	X =  365.642  mm,	Y =   -78.945  mm,	Z =   -251.457  mm,
	W =  90.000 deg,	P =   0.000 deg,	R =   90.000 deg
};
P[3235]{
   GP1:
	UF : 0, UT : 6,		CONFIG : 'N U T, 0, 0, 0',
	X =  364.632  mm,	Y =   -78.307  mm,	Z =   -251.452  mm,
	W =  90.000 deg,	P =   0.000 deg,	R =   90.000 deg
};
P[3236]{
   GP1:
	UF : 0, UT : 6,		CONFIG : 'N U T, 0, 0, 0',
	X =  359.937  mm,	Y =   -76.604  mm,	Z =   -251.287  mm,
	W =  90.000 deg,	P =   0.000 deg,	R =   90.000 deg
};
P[3237]{
   GP1:
	UF : 0, UT : 6,		CONFIG : 'N U T, 0, 0, 0',
	X =  357.838  mm,	Y =   -76.355  mm,	Z =   -251.028  mm,
	W =  90.000 deg,	P =   0.000 deg,	R =   90.000 deg
};
P[3238]{
   GP1:
	UF : 0, UT : 6,		CONFIG : 'N U T, 0, 0, 0',
	X =  355.930  mm,	Y =   -76.626  mm,	Z =   -251.285  mm,
	W =  90.000 deg,	P =   0.000 deg,	R =   90.000 deg
};
P[3239]{
   GP1:
	UF : 0, UT : 6,		CONFIG : 'N U T, 0, 0, 0',
	X =  353.780  mm,	Y =   -77.047  mm,	Z =   -251.080  mm,
	W =  90.000 deg,	P =   0.000 deg,	R =   90.000 deg
};
P[3240]{
   GP1:
	UF : 0, UT : 6,		CONFIG : 'N U T, 0, 0, 0',
	X =  353.192  mm,	Y =   -77.362  mm,	Z =   -251.275  mm,
	W =  90.000 deg,	P =   0.000 deg,	R =   90.000 deg
};
P[3241]{
   GP1:
	UF : 0, UT : 6,		CONFIG : 'N U T, 0, 0, 0',
	X =  352.107  mm,	Y =   -77.912  mm,	Z =   -251.405  mm,
	W =  90.000 deg,	P =   0.000 deg,	R =   90.000 deg
};
P[3242]{
   GP1:
	UF : 0, UT : 6,		CONFIG : 'N U T, 0, 0, 0',
	X =  349.503  mm,	Y =   -79.254  mm,	Z =   -251.336  mm,
	W =  90.000 deg,	P =   0.000 deg,	R =   90.000 deg
};
P[3243]{
   GP1:
	UF : 0, UT : 6,		CONFIG : 'N U T, 0, 0, 0',
	X =  346.830  mm,	Y =   -80.833  mm,	Z =   -251.422  mm,
	W =  90.000 deg,	P =   0.000 deg,	R =   90.000 deg
};
P[3244]{
   GP1:
	UF : 0, UT : 6,		CONFIG : 'N U T, 0, 0, 0',
	X =  345.177  mm,	Y =   -81.811  mm,	Z =   -251.480  mm,
	W =  90.000 deg,	P =   0.000 deg,	R =   90.000 deg
};
P[3245]{
   GP1:
	UF : 0, UT : 6,		CONFIG : 'N U T, 0, 0, 0',
	X =  342.562  mm,	Y =   -83.180  mm,	Z =   -251.136  mm,
	W =  90.000 deg,	P =   0.000 deg,	R =   90.000 deg
};
P[3246]{
   GP1:
	UF : 0, UT : 6,		CONFIG : 'N U T, 0, 0, 0',
	X =  337.354  mm,	Y =   -86.298  mm,	Z =   -251.409  mm,
	W =  90.000 deg,	P =   0.000 deg,	R =   90.000 deg
};
P[3247]{
   GP1:
	UF : 0, UT : 6,		CONFIG : 'N U T, 0, 0, 0',
	X =  336.571  mm,	Y =   -86.625  mm,	Z =   -251.103  mm,
	W =  90.000 deg,	P =   0.000 deg,	R =   90.000 deg
};
P[3248]{
   GP1:
	UF : 0, UT : 6,		CONFIG : 'N U T, 0, 0, 0',
	X =  335.626  mm,	Y =   -87.310  mm,	Z =   -251.441  mm,
	W =  90.000 deg,	P =   0.000 deg,	R =   90.000 deg
};
P[3249]{
   GP1:
	UF : 0, UT : 6,		CONFIG : 'N U T, 0, 0, 0',
	X =  334.747  mm,	Y =   -87.679  mm,	Z =   -251.108  mm,
	W =  90.000 deg,	P =   0.000 deg,	R =   90.000 deg
};
P[3250]{
   GP1:
	UF : 0, UT : 6,		CONFIG : 'N U T, 0, 0, 0',
	X =  332.760  mm,	Y =   -88.868  mm,	Z =   -251.208  mm,
	W =  90.000 deg,	P =   0.000 deg,	R =   90.000 deg
};
P[3251]{
   GP1:
	UF : 0, UT : 6,		CONFIG : 'N U T, 0, 0, 0',
	X =  332.024  mm,	Y =   -89.291  mm,	Z =   -251.201  mm,
	W =  90.000 deg,	P =   0.000 deg,	R =   90.000 deg
};
P[3252]{
   GP1:
	UF : 0, UT : 6,		CONFIG : 'N U T, 0, 0, 0',
	X =  326.457  mm,	Y =   -92.567  mm,	Z =   -251.352  mm,
	W =  90.000 deg,	P =   0.000 deg,	R =   90.000 deg
};
P[3253]{
   GP1:
	UF : 0, UT : 6,		CONFIG : 'N U T, 0, 0, 0',
	X =  323.513  mm,	Y =   -94.171  mm,	Z =   -251.117  mm,
	W =  90.000 deg,	P =   0.000 deg,	R =   90.000 deg
};
P[3254]{
   GP1:
	UF : 0, UT : 6,		CONFIG : 'N U T, 0, 0, 0',
	X =  318.378  mm,	Y =   -97.275  mm,	Z =   -251.456  mm,
	W =  90.000 deg,	P =   0.000 deg,	R =   90.000 deg
};
P[3255]{
   GP1:
	UF : 0, UT : 6,		CONFIG : 'N U T, 0, 0, 0',
	X =  317.185  mm,	Y =   -97.859  mm,	Z =   -251.203  mm,
	W =  90.000 deg,	P =   0.000 deg,	R =   90.000 deg
};
P[3256]{
   GP1:
	UF : 0, UT : 6,		CONFIG : 'N U T, 0, 0, 0',
	X =  316.114  mm,	Y =   -98.543  mm,	Z =   -251.361  mm,
	W =  90.000 deg,	P =   0.000 deg,	R =   90.000 deg
};
P[3257]{
   GP1:
	UF : 0, UT : 6,		CONFIG : 'N U T, 0, 0, 0',
	X =  314.155  mm,	Y =   -99.553  mm,	Z =   -251.068  mm,
	W =  90.000 deg,	P =   0.000 deg,	R =   90.000 deg
};
P[3258]{
   GP1:
	UF : 0, UT : 6,		CONFIG : 'N U T, 0, 0, 0',
	X =  313.148  mm,	Y =   -100.225  mm,	Z =   -251.288  mm,
	W =  90.000 deg,	P =   0.000 deg,	R =   90.000 deg
};
P[3259]{
   GP1:
	UF : 0, UT : 6,		CONFIG : 'N U T, 0, 0, 0',
	X =  310.503  mm,	Y =   -101.793  mm,	Z =   -251.386  mm,
	W =  90.000 deg,	P =   0.000 deg,	R =   90.000 deg
};
P[3260]{
   GP1:
	UF : 0, UT : 6,		CONFIG : 'N U T, 0, 0, 0',
	X =  309.548  mm,	Y =   -102.306  mm,	Z =   -251.294  mm,
	W =  90.000 deg,	P =   0.000 deg,	R =   90.000 deg
};
P[3261]{
   GP1:
	UF : 0, UT : 6,		CONFIG : 'N U T, 0, 0, 0',
	X =  306.446  mm,	Y =   -104.089  mm,	Z =   -251.273  mm,
	W =  90.000 deg,	P =   0.000 deg,	R =   90.000 deg
};
P[3262]{
   GP1:
	UF : 0, UT : 6,		CONFIG : 'N U T, 0, 0, 0',
	X =  303.476  mm,	Y =   -105.784  mm,	Z =   -251.224  mm,
	W =  90.000 deg,	P =   0.000 deg,	R =   90.000 deg
};
P[3263]{
   GP1:
	UF : 0, UT : 6,		CONFIG : 'N U T, 0, 0, 0',
	X =  302.259  mm,	Y =   -106.421  mm,	Z =   -251.065  mm,
	W =  90.000 deg,	P =   0.000 deg,	R =   90.000 deg
};
P[3264]{
   GP1:
	UF : 0, UT : 6,		CONFIG : 'N U T, 0, 0, 0',
	X =  301.391  mm,	Y =   -107.018  mm,	Z =   -251.300  mm,
	W =  90.000 deg,	P =   0.000 deg,	R =   90.000 deg
};
P[3265]{
   GP1:
	UF : 0, UT : 6,		CONFIG : 'N U T, 0, 0, 0',
	X =  298.634  mm,	Y =   -108.624  mm,	Z =   -251.331  mm,
	W =  90.000 deg,	P =   0.000 deg,	R =   90.000 deg
};
P[3266]{
   GP1:
	UF : 0, UT : 6,		CONFIG : 'N U T, 0, 0, 0',
	X =  297.240  mm,	Y =   -109.333  mm,	Z =   -251.101  mm,
	W =  90.000 deg,	P =   0.000 deg,	R =   90.000 deg
};
P[3267]{
   GP1:
	UF : 0, UT : 6,		CONFIG : 'N U T, 0, 0, 0',
	X =  295.855  mm,	Y =   -110.282  mm,	Z =   -251.463  mm,
	W =  90.000 deg,	P =   0.000 deg,	R =   90.000 deg
};
P[3268]{
   GP1:
	UF : 0, UT : 6,		CONFIG : 'N U T, 0, 0, 0',
	X =  295.155  mm,	Y =   -110.620  mm,	Z =   -251.300  mm,
	W =  90.000 deg,	P =   0.000 deg,	R =   90.000 deg
};
P[3269]{
   GP1:
	UF : 0, UT : 6,		CONFIG : 'N U T, 0, 0, 0',
	X =  294.447  mm,	Y =   -111.014  mm,	Z =   -251.266  mm,
	W =  90.000 deg,	P =   0.000 deg,	R =   90.000 deg
};
P[3270]{
   GP1:
	UF : 0, UT : 6,		CONFIG : 'N U T, 0, 0, 0',
	X =  293.600  mm,	Y =   -111.593  mm,	Z =   -251.484  mm,
	W =  90.000 deg,	P =   0.000 deg,	R =   90.000 deg
};
P[3271]{
   GP1:
	UF : 0, UT : 6,		CONFIG : 'N U T, 0, 0, 0',
	X =  291.360  mm,	Y =   -112.706  mm,	Z =   -251.045  mm,
	W =  90.000 deg,	P =   0.000 deg,	R =   90.000 deg
};
P[3272]{
   GP1:
	UF : 0, UT : 6,		CONFIG : 'N U T, 0, 0, 0',
	X =  289.173  mm,	Y =   -114.076  mm,	Z =   -251.307  mm,
	W =  90.000 deg,	P =   0.000 deg,	R =   90.000 deg
};
P[3273]{
   GP1:
	UF : 0, UT : 6,		CONFIG : 'N U T, 0, 0, 0',
	X =  287.782  mm,	Y =   -114.866  mm,	Z =   -251.275  mm,
	W =  90.000 deg,	P =   0.000 deg,	R =   90.000 deg
};
P[3274]{
   GP1:
	UF : 0, UT : 6,		CONFIG : 'N U T, 0, 0, 0',
	X =  285.771  mm,	Y =   -116.071  mm,	Z =   -251.381  mm,
	W =  90.000 deg,	P =   0.000 deg,	R =   90.000 deg
};
P[3275]{
   GP1:
	UF : 0, UT : 6,		CONFIG : 'N U T, 0, 0, 0',
	X =  283.058  mm,	Y =   -117.627  mm,	Z =   -251.356  mm,
	W =  90.000 deg,	P =   0.000 deg,	R =   90.000 deg
};
P[3276]{
   GP1:
	UF : 0, UT : 6,		CONFIG : 'N U T, 0, 0, 0',
	X =  282.254  mm,	Y =   -118.089  mm,	Z =   -251.350  mm,
	W =  90.000 deg,	P =   0.000 deg,	R =   90.000 deg
};
P[3277]{
   GP1:
	UF : 0, UT : 6,		CONFIG : 'N U T, 0, 0, 0',
	X =  279.242  mm,	Y =   -119.866  mm,	Z =   -251.442  mm,
	W =  90.000 deg,	P =   0.000 deg,	R =   90.000 deg
};
P[3278]{
   GP1:
	UF : 0, UT : 6,		CONFIG : 'N U T, 0, 0, 0',
	X =  277.448  mm,	Y =   -120.879  mm,	Z =   -251.386  mm,
	W =  90.000 deg,	P =   0.000 deg,	R =   90.000 deg
};
P[3279]{
   GP1:
	UF : 0, UT : 6,		CONFIG : 'N U T, 0, 0, 0',
	X =  276.850  mm,	Y =   -121.103  mm,	Z =   -251.091  mm,
	W =  90.000 deg,	P =   0.000 deg,	R =   90.000 deg
};
P[3280]{
   GP1:
	UF : 0, UT : 6,		CONFIG : 'N U T, 0, 0, 0',
	X =  275.892  mm,	Y =   -121.675  mm,	Z =   -251.138  mm,
	W =  90.000 deg,	P =   0.000 deg,	R =   90.000 deg
};
P[3281]{
   GP1:
	UF : 0, UT : 6,		CONFIG : 'N U T, 0, 0, 0',
	X =  272.785  mm,	Y =   -123.489  mm,	Z =   -251.187  mm,
	W =  90.000 deg,	P =   0.000 deg,	R =   90.000 deg
};
P[3282]{
   GP1:
	UF : 0, UT : 6,		CONFIG : 'N U T, 0, 0, 0',
	X =  270.250  mm,	Y =   -124.968  mm,	Z =   -251.224  mm,
	W =  90.000 deg,	P =   0.000 deg,	R =   90.000 deg
};
P[3283]{
   GP1:
	UF : 0, UT : 6,		CONFIG : 'N U T, 0, 0, 0',
	X =  267.856  mm,	Y =   -126.325  mm,	Z =   -251.164  mm,
	W =  90.000 deg,	P =   0.000 deg,	R =   90.000 deg
};
P[3284]{
   GP1:
	UF : 0, UT : 6,		CONFIG : 'N U T, 0, 0, 0',
	X =  266.892  mm,	Y =   -126.881  mm,	Z =   -251.161  mm,
	W =  90.000 deg,	P =   0.000 deg,	R =   90.000 deg
};
P[3285]{
   GP1:
	UF : 0, UT : 6,		CONFIG : 'N U T, 0, 0, 0',
	X =  265.651  mm,	Y =   -127.610  mm,	Z =   -251.192  mm,
	W =  90.000 deg,	P =   0.000 deg,	R =   90.000 deg
};
P[3286]{
   GP1:
	UF : 0, UT : 6,		CONFIG : 'N U T, 0, 0, 0',
	X =  262.122  mm,	Y =   -129.745  mm,	Z =   -251.428  mm,
	W =  90.000 deg,	P =   0.000 deg,	R =   90.000 deg
};
P[3287]{
   GP1:
	UF : 0, UT : 6,		CONFIG : 'N U T, 0, 0, 0',
	X =  257.854  mm,	Y =   -132.149  mm,	Z =   -251.281  mm,
	W =  90.000 deg,	P =   0.000 deg,	R =   90.000 deg
};
P[3288]{
   GP1:
	UF : 0, UT : 6,		CONFIG : 'N U T, 0, 0, 0',
	X =  256.892  mm,	Y =   -132.728  mm,	Z =   -251.340  mm,
	W =  90.000 deg,	P =   0.000 deg,	R =   90.000 deg
};
P[3289]{
   GP1:
	UF : 0, UT : 6,		CONFIG : 'N U T, 0, 0, 0',
	X =  256.166  mm,	Y =   -133.205  mm,	Z =   -251.481  mm,
	W =  90.000 deg,	P =   0.000 deg,	R =   90.000 deg
};
P[3290]{
   GP1:
	UF : 0, UT : 6,		CONFIG : 'N U T, 0, 0, 0',
	X =  251.767  mm,	Y =   -135.749  mm,	Z =   -251.492  mm,
	W =  90.000 deg,	P =   0.000 deg,	R =   90.000 deg
};
P[3291]{
   GP1:
	UF : 0, UT : 6,		CONFIG : 'N U T, 0, 0, 0',
	X =  249.950  mm,	Y =   -136.758  mm,	Z =   -251.391  mm,
	W =  90.000 deg,	P =   0.000 deg,	R =   90.000 deg
};
P[3292]{
   GP1:
	UF : 0, UT : 6,		CONFIG : 'N U T, 0, 0, 0',
	X =  248.916  mm,	Y =   -137.229  mm,	Z =   -251.087  mm,
	W =  90.000 deg,	P =   0.000 deg,	R =   90.000 deg
};
P[3293]{
   GP1:
	UF : 0, UT : 6,		CONFIG : 'N U T, 0, 0, 0',
	X =  244.453  mm,	Y =   -139.858  mm,	Z =   -251.213  mm,
	W =  90.000 deg,	P =   0.000 deg,	R =   90.000 deg
};
P[3294]{
   GP1:
	UF : 0, UT : 6,		CONFIG : 'N U T, 0, 0, 0',
	X =  241.068  mm,	Y =   -141.906  mm,	Z =   -251.440  mm,
	W =  90.000 deg,	P =   0.000 deg,	R =   90.000 deg
};
P[3295]{
   GP1:
	UF : 0, UT : 6,		CONFIG : 'N U T, 0, 0, 0',
	X =  239.719  mm,	Y =   -142.513  mm,	Z =   -251.022  mm,
	W =  90.000 deg,	P =   0.000 deg,	R =   90.000 deg
};
P[3296]{
   GP1:
	UF : 0, UT : 6,		CONFIG : 'N U T, 0, 0, 0',
	X =  234.349  mm,	Y =   -145.704  mm,	Z =   -251.240  mm,
	W =  90.000 deg,	P =   0.000 deg,	R =   90.000 deg
};
P[3297]{
   GP1:
	UF : 0, UT : 6,		CONFIG : 'N U T, 0, 0, 0',
	X =  230.397  mm,	Y =   -148.015  mm,	Z =   -251.313  mm,
	W =  90.000 deg,	P =   0.000 deg,	R =   90.000 deg
};
P[3298]{
   GP1:
	UF : 0, UT : 6,		CONFIG : 'N U T, 0, 0, 0',
	X =  229.049  mm,	Y =   -148.679  mm,	Z =   -251.034  mm,
	W =  90.000 deg,	P =   0.000 deg,	R =   90.000 deg
};
P[3299]{
   GP1:
	UF : 0, UT : 6,		CONFIG : 'N U T, 0, 0, 0',
	X =  226.182  mm,	Y =   -150.383  mm,	Z =   -251.153  mm,
	W =  90.000 deg,	P =   0.000 deg,	R =   90.000 deg
};
P[3300]{
   GP1:
	UF : 0, UT : 6,		CONFIG : 'N U T, 0, 0, 0',
	X =  222.300  mm,	Y =   -152.731  mm,	Z =   -251.410  mm,
	W =  90.000 deg,	P =   0.000 deg,	R =   90.000 deg
};
P[3301]{
   GP1:
	UF : 0, UT : 6,		CONFIG : 'N U T, 0, 0, 0',
	X =  220.364  mm,	Y =   -153.720  mm,	Z =   -251.098  mm,
	W =  90.000 deg,	P =   0.000 deg,	R =   90.000 deg
};
P[3302]{
   GP1:
	UF : 0, UT : 6,		CONFIG : 'N U T, 0, 0, 0',
	X =  218.957  mm,	Y =   -154.647  mm,	Z =   -251.377  mm,
	W =  90.000 deg,	P =   0.000 deg,	R =   90.000 deg
};
P[3303]{
   GP1:
	UF : 0, UT : 6,		CONFIG : 'N U T, 0, 0, 0',
	X =  214.839  mm,	Y =   -156.990  mm,	Z =   -251.293  mm,
	W =  90.000 deg,	P =   0.000 deg,	R =   90.000 deg
};
P[3304]{
   GP1:
	UF : 0, UT : 6,		CONFIG : 'N U T, 0, 0, 0',
	X =  213.334  mm,	Y =   -157.757  mm,	Z =   -251.045  mm,
	W =  90.000 deg,	P =   0.000 deg,	R =   90.000 deg
};
P[3305]{
   GP1:
	UF : 0, UT : 6,		CONFIG : 'N U T, 0, 0, 0',
	X =  209.437  mm,	Y =   -160.137  mm,	Z =   -251.362  mm,
	W =  90.000 deg,	P =   0.000 deg,	R =   90.000 deg
};
P[3306]{
   GP1:
	UF : 0, UT : 6,		CONFIG : 'N U T, 0, 0, 0',
	X =  205.579  mm,	Y =   -162.285  mm,	Z =   -251.166  mm,
	W =  90.000 deg,	P =   0.000 deg,	R =   90.000 deg
};
P[3307]{
   GP1:
	UF : 0, UT : 6,		CONFIG : 'N U T, 0, 0, 0',
	X =  204.500  mm,	Y =   -163.043  mm,	Z =   -251.494  mm,
	W =  90.000 deg,	P =   0.000 deg,	R =   90.000 deg
};
P[3308]{
   GP1:
	UF : 0, UT : 6,		CONFIG : 'N U T, 0, 0, 0',
	X =  203.455  mm,	Y =   -163.573  mm,	Z =   -251.316  mm,
	W =  90.000 deg,	P =   0.000 deg,	R =   90.000 deg
};
P[3309]{
   GP1:
	UF : 0, UT : 6,		CONFIG : 'N U T, 0, 0, 0',
	X =  202.079  mm,	Y =   -164.250  mm,	Z =   -251.032  mm,
	W =  90.000 deg,	P =   0.000 deg,	R =   90.000 deg
};
P[3310]{
   GP1:
	UF : 0, UT : 6,		CONFIG : 'N U T, 0, 0, 0',
	X =  199.549  mm,	Y =   -165.840  mm,	Z =   -251.344  mm,
	W =  90.000 deg,	P =   0.000 deg,	R =   90.000 deg
};
P[3311]{
   GP1:
	UF : 0, UT : 6,		CONFIG : 'N U T, 0, 0, 0',
	X =  197.860  mm,	Y =   -166.804  mm,	Z =   -251.317  mm,
	W =  90.000 deg,	P =   0.000 deg,	R =   90.000 deg
};
P[3312]{
   GP1:
	UF : 0, UT : 6,		CONFIG : 'N U T, 0, 0, 0',
	X =  196.154  mm,	Y =   -167.750  mm,	Z =   -251.223  mm,
	W =  90.000 deg,	P =   0.000 deg,	R =   90.000 deg
};
P[3313]{
   GP1:
	UF : 0, UT : 6,		CONFIG : 'N U T, 0, 0, 0',
	X =  193.452  mm,	Y =   -169.373  mm,	Z =   -251.377  mm,
	W =  90.000 deg,	P =   0.000 deg,	R =   90.000 deg
};
P[3314]{
   GP1:
	UF : 0, UT : 6,		CONFIG : 'N U T, 0, 0, 0',
	X =  192.530  mm,	Y =   -169.912  mm,	Z =   -251.393  mm,
	W =  90.000 deg,	P =   0.000 deg,	R =   90.000 deg
};
P[3315]{
   GP1:
	UF : 0, UT : 6,		CONFIG : 'N U T, 0, 0, 0',
	X =  189.367  mm,	Y =   -171.663  mm,	Z =   -251.212  mm,
	W =  90.000 deg,	P =   0.000 deg,	R =   90.000 deg
};
P[3316]{
   GP1:
	UF : 0, UT : 6,		CONFIG : 'N U T, 0, 0, 0',
	X =  188.461  mm,	Y =   -172.307  mm,	Z =   -251.503  mm,
	W =  90.000 deg,	P =   0.000 deg,	R =   90.000 deg
};
P[3317]{
   GP1:
	UF : 0, UT : 6,		CONFIG : 'N U T, 0, 0, 0',
	X =  184.461  mm,	Y =   -174.616  mm,	Z =   -251.502  mm,
	W =  90.000 deg,	P =   0.000 deg,	R =   90.000 deg
};
P[3318]{
   GP1:
	UF : 0, UT : 6,		CONFIG : 'N U T, 0, 0, 0',
	X =  183.601  mm,	Y =   -175.029  mm,	Z =   -251.299  mm,
	W =  90.000 deg,	P =   0.000 deg,	R =   90.000 deg
};
P[3319]{
   GP1:
	UF : 0, UT : 6,		CONFIG : 'N U T, 0, 0, 0',
	X =  180.948  mm,	Y =   -176.632  mm,	Z =   -251.473  mm,
	W =  90.000 deg,	P =   0.000 deg,	R =   90.000 deg
};
P[3320]{
   GP1:
	UF : 0, UT : 6,		CONFIG : 'N U T, 0, 0, 0',
	X =  179.809  mm,	Y =   -177.300  mm,	Z =   -251.496  mm,
	W =  90.000 deg,	P =   0.000 deg,	R =   90.000 deg
};
P[3321]{
   GP1:
	UF : 0, UT : 6,		CONFIG : 'N U T, 0, 0, 0',
	X =  178.979  mm,	Y =   -177.755  mm,	Z =   -251.439  mm,
	W =  90.000 deg,	P =   0.000 deg,	R =   90.000 deg
};
P[3322]{
   GP1:
	UF : 0, UT : 6,		CONFIG : 'N U T, 0, 0, 0',
	X =  177.248  mm,	Y =   -178.708  mm,	Z =   -251.325  mm,
	W =  90.000 deg,	P =   0.000 deg,	R =   90.000 deg
};
P[3323]{
   GP1:
	UF : 0, UT : 6,		CONFIG : 'N U T, 0, 0, 0',
	X =  173.062  mm,	Y =   -181.196  mm,	Z =   -251.498  mm,
	W =  90.000 deg,	P =   0.000 deg,	R =   90.000 deg
};
P[3324]{
   GP1:
	UF : 0, UT : 6,		CONFIG : 'N U T, 0, 0, 0',
	X =  169.773  mm,	Y =   -183.093  mm,	Z =   -251.493  mm,
	W =  90.000 deg,	P =   0.000 deg,	R =   90.000 deg
};
P[3325]{
   GP1:
	UF : 0, UT : 6,		CONFIG : 'N U T, 0, 0, 0',
	X =  168.501  mm,	Y =   -183.759  mm,	Z =   -251.324  mm,
	W =  90.000 deg,	P =   0.000 deg,	R =   90.000 deg
};
P[3326]{
   GP1:
	UF : 0, UT : 6,		CONFIG : 'N U T, 0, 0, 0',
	X =  167.751  mm,	Y =   -184.156  mm,	Z =   -251.239  mm,
	W =  90.000 deg,	P =   0.000 deg,	R =   90.000 deg
};
P[3327]{
   GP1:
	UF : 0, UT : 6,		CONFIG : 'N U T, 0, 0, 0',
	X =  166.575  mm,	Y =   -184.935  mm,	Z =   -251.482  mm,
	W =  90.000 deg,	P =   0.000 deg,	R =   90.000 deg
};
P[3328]{
   GP1:
	UF : 0, UT : 6,		CONFIG : 'N U T, 0, 0, 0',
	X =  159.993  mm,	Y =   -188.722  mm,	Z =   -251.449  mm,
	W =  90.000 deg,	P =   0.000 deg,	R =   90.000 deg
};
P[3329]{
   GP1:
	UF : 0, UT : 6,		CONFIG : 'N U T, 0, 0, 0',
	X =  156.405  mm,	Y =   -190.684  mm,	Z =   -251.183  mm,
	W =  90.000 deg,	P =   0.000 deg,	R =   90.000 deg
};
P[3330]{
   GP1:
	UF : 0, UT : 6,		CONFIG : 'N U T, 0, 0, 0',
	X =  155.527  mm,	Y =   -191.243  mm,	Z =   -251.310  mm,
	W =  90.000 deg,	P =   0.000 deg,	R =   90.000 deg
};
P[3331]{
   GP1:
	UF : 0, UT : 6,		CONFIG : 'N U T, 0, 0, 0',
	X =  154.467  mm,	Y =   -191.889  mm,	Z =   -251.392  mm,
	W =  90.000 deg,	P =   0.000 deg,	R =   90.000 deg
};
P[3332]{
   GP1:
	UF : 0, UT : 6,		CONFIG : 'N U T, 0, 0, 0',
	X =  153.561  mm,	Y =   -192.345  mm,	Z =   -251.228  mm,
	W =  90.000 deg,	P =   0.000 deg,	R =   90.000 deg
};
P[3333]{
   GP1:
	UF : 0, UT : 6,		CONFIG : 'N U T, 0, 0, 0',
	X =  151.064  mm,	Y =   -193.853  mm,	Z =   -251.389  mm,
	W =  90.000 deg,	P =   0.000 deg,	R =   90.000 deg
};
P[3334]{
   GP1:
	UF : 0, UT : 6,		CONFIG : 'N U T, 0, 0, 0',
	X =  149.622  mm,	Y =   -194.718  mm,	Z =   -251.468  mm,
	W =  90.000 deg,	P =   0.000 deg,	R =   90.000 deg
};
P[3335]{
   GP1:
	UF : 0, UT : 6,		CONFIG : 'N U T, 0, 0, 0',
	X =  147.531  mm,	Y =   -195.898  mm,	Z =   -251.400  mm,
	W =  90.000 deg,	P =   0.000 deg,	R =   90.000 deg
};
P[3336]{
   GP1:
	UF : 0, UT : 6,		CONFIG : 'N U T, 0, 0, 0',
	X =  146.000  mm,	Y =   -196.707  mm,	Z =   -251.220  mm,
	W =  90.000 deg,	P =   0.000 deg,	R =   90.000 deg
};
P[3337]{
   GP1:
	UF : 0, UT : 6,		CONFIG : 'N U T, 0, 0, 0',
	X =  144.867  mm,	Y =   -197.415  mm,	Z =   -251.350  mm,
	W =  90.000 deg,	P =   0.000 deg,	R =   90.000 deg
};
P[3338]{
   GP1:
	UF : 0, UT : 6,		CONFIG : 'N U T, 0, 0, 0',
	X =  141.987  mm,	Y =   -199.098  mm,	Z =   -251.400  mm,
	W =  90.000 deg,	P =   0.000 deg,	R =   90.000 deg
};
P[3339]{
   GP1:
	UF : 0, UT : 6,		CONFIG : 'N U T, 0, 0, 0',
	X =  141.039  mm,	Y =   -199.684  mm,	Z =   -251.492  mm,
	W =  90.000 deg,	P =   0.000 deg,	R =   90.000 deg
};
P[3340]{
   GP1:
	UF : 0, UT : 6,		CONFIG : 'N U T, 0, 0, 0',
	X =  139.194  mm,	Y =   -200.553  mm,	Z =   -251.017  mm,
	W =  90.000 deg,	P =   0.000 deg,	R =   90.000 deg
};
P[3341]{
   GP1:
	UF : 0, UT : 6,		CONFIG : 'N U T, 0, 0, 0',
	X =  137.043  mm,	Y =   -201.854  mm,	Z =   -251.159  mm,
	W =  90.000 deg,	P =   0.000 deg,	R =   90.000 deg
};
P[3342]{
   GP1:
	UF : 0, UT : 6,		CONFIG : 'N U T, 0, 0, 0',
	X =  135.134  mm,	Y =   -202.930  mm,	Z =   -251.096  mm,
	W =  90.000 deg,	P =   0.000 deg,	R =   90.000 deg
};
P[3343]{
   GP1:
	UF : 0, UT : 6,		CONFIG : 'N U T, 0, 0, 0',
	X =  133.307  mm,	Y =   -204.097  mm,	Z =   -251.370  mm,
	W =  90.000 deg,	P =   0.000 deg,	R =   90.000 deg
};
P[3344]{
   GP1:
	UF : 0, UT : 6,		CONFIG : 'N U T, 0, 0, 0',
	X =  129.302  mm,	Y =   -206.469  mm,	Z =   -251.512  mm,
	W =  90.000 deg,	P =   0.000 deg,	R =   90.000 deg
};
P[3345]{
   GP1:
	UF : 0, UT : 6,		CONFIG : 'N U T, 0, 0, 0',
	X =  127.360  mm,	Y =   -207.438  mm,	Z =   -251.141  mm,
	W =  90.000 deg,	P =   0.000 deg,	R =   90.000 deg
};
P[3346]{
   GP1:
	UF : 0, UT : 6,		CONFIG : 'N U T, 0, 0, 0',
	X =  126.300  mm,	Y =   -208.144  mm,	Z =   -251.372  mm,
	W =  90.000 deg,	P =   0.000 deg,	R =   90.000 deg
};
P[3347]{
   GP1:
	UF : 0, UT : 6,		CONFIG : 'N U T, 0, 0, 0',
	X =  124.357  mm,	Y =   -209.289  mm,	Z =   -251.427  mm,
	W =  90.000 deg,	P =   0.000 deg,	R =   90.000 deg
};
P[3348]{
   GP1:
	UF : 0, UT : 6,		CONFIG : 'N U T, 0, 0, 0',
	X =  122.937  mm,	Y =   -210.015  mm,	Z =   -251.199  mm,
	W =  90.000 deg,	P =   0.000 deg,	R =   90.000 deg
};
P[3349]{
   GP1:
	UF : 0, UT : 6,		CONFIG : 'N U T, 0, 0, 0',
	X =  119.572  mm,	Y =   -212.010  mm,	Z =   -251.327  mm,
	W =  90.000 deg,	P =   0.000 deg,	R =   90.000 deg
};
P[3350]{
   GP1:
	UF : 0, UT : 6,		CONFIG : 'N U T, 0, 0, 0',
	X =  210.000  mm,	Y =   -375.000  mm,	Z =   -250.000  mm,
	W =  90.000 deg,	P =   0.000 deg,	R =   90.000 deg
};
/END
